FUNCTION "TE-SS" : VOID	// FC 11
AUTHOR : SIMATIC
FAMILY : EA_DIS
NAME : TE_SS
VERSION : 3.0
BEGIN
// (block stored without names or comments; labels and parameter names are numbered)
NETWORK
TITLE =
      L     0;
      L     #PARAM22;
      ==I;
      JC    M001;
      T     MW 214;
      L     MB 214;
      T     LW 10;
      OPN   DB [LW 10];
      L     MB 215;
      SLW   3;
      LAR1;
      L     DBW [AR1,P#0.0];
      T     MB 227;
M001: L     #PARAM20;
      T     MW 214;
      L     MB 214;
      T     LW 10;
      OPN   DB [LW 10];
      L     #PARAM20;
      T     MW 214;
      L     MB 215;
      SLW   3;
      LAR1;
      L     DBW [AR1,P#0.0];
      T     MW 200;
      L     DBW [AR1,P#2.0];
      T     MW 202;
      L     DBW [AR1,P#4.0];
      T     MW 204;
      L     DBW [AR1,P#10.0];
      T     MW 208;
      L     DBW [AR1,P#12.0];
      T     MW 210;
      L     DBW [AR1,P#14.0];
      T     MW 212;
      L     DBW [AR1,P#16.0];
      T     MW 206;
      A     #PARAM1;
      A     M 204.7;
      =     M 203.2;
      A     #PARAM1;
      AN    M 204.7;
      =     M 202.0;
      A     #PARAM2;
      =     M 202.1;
      A     #PARAM3;
      AN    M 203.3;
      =     M 211.5;
      A     #PARAM3;
      =     M 203.3;
      A     #PARAM4;
      AN    M 203.0;
      =     M 211.7;
      A     #PARAM4;
      =     M 203.0;
      A     #PARAM8;
      AN    M 203.1;
      =     M 211.6;
      A     #PARAM8;
      =     M 203.1;
      A     #PARAM9;
      AN    M 203.4;
      =     M 211.4;
      A     #PARAM9;
      =     M 203.4;
      A     #PARAM10;
      =     M 202.2;
      A     #PARAM11;
      =     M 203.5;
      A     #PARAM7;
      =     M 213.0;
      A     #PARAM6;
      =     M 210.1;
      A     #PARAM13;
      =     M 210.7;
      A     #PARAM14;
      =     M 210.6;
      A     #PARAM15;
      =     M 210.5;
      A     #PARAM16;
      =     M 210.4;
      A     #PARAM17;
      =     M 210.3;
      A     #PARAM18;
      =     M 210.2;
      A     #PARAM19;
      =     M 200.4;
      A     #PARAM12;
      =     M 210.0;
      A     #PARAM5;
      =     M 203.6;
NETWORK
TITLE =
      A     M 210.7;
      AN    M 210.6;
      =     M 212.7;
      AN    M 210.7;
      A     M 210.6;
      =     M 212.5;
      A     M 210.5;
      AN    M 210.4;
      =     M 212.6;
      AN    M 210.5;
      A     M 210.4;
      =     M 212.4;
NETWORK
TITLE =
      A     M 227.3;
      AN    M 202.5;
      =     M 211.3;
      A     M 227.3;
      =     M 202.5;
      A     M 227.2;
      AN    M 202.6;
      =     M 211.2;
      A     M 227.2;
      =     M 202.6;
NETWORK
TITLE =
      A     M 203.1;
      A     M 210.1;
      AN    M 203.0;
      AN    M 203.6;
      =     M 218.7;
      A     M 203.0;
      A     M 210.1;
      AN    M 203.6;
      =     M 219.7;
      A     M 227.2;
      A     M 227.1;
      AN    M 227.3;
      AN    M 227.0;
      AN    M 219.7;
      AN    M 203.6;
      =     M 218.5;
      A     M 227.3;
      A     M 227.1;
      AN    M 227.0;
      AN    M 218.7;
      AN    M 203.6;
      =     M 219.5;
      A     M 203.4;
      AN    M 203.3;
      AN    M 219.7;
      AN    M 203.6;
      AN    M 227.0;
      AN    M 219.5;
      =     M 218.3;
      A     M 203.3;
      AN    M 218.7;
      AN    M 218.5;
      AN    M 203.6;
      AN    M 227.0;
      =     M 219.3;
      A     M 218.7;
      O     M 218.5;
      O     M 218.3;
      =     M 212.3;
      A     M 219.7;
      O     M 219.5;
      O     M 219.3;
      =     M 212.1;
      A     M 211.6;
      A     M 218.7;
      O;
      A     M 211.2;
      A     M 218.5;
      O;
      A     M 211.4;
      A     M 218.3;
      =     M 212.2;
      A     M 211.7;
      A     M 219.7;
      O;
      A     M 211.3;
      A     M 219.5;
      O;
      A     M 211.5;
      A     M 219.3;
      =     M 212.0;
NETWORK
TITLE =
      A     M 211.6;
      O     M 211.2;
      =     M 213.4;
      A     M 211.7;
      O     M 211.3;
      =     M 213.5;
      A     M 203.6;
      O     M 227.0;
      =     M 213.7;
NETWORK
TITLE =
      A     M 212.7;
      O     M 213.7;
      O     M 212.3;
      R     M 211.1;
      R     M 211.0;
      A     M 203.2;
      S     M 211.1;
      A     M 202.0;
      S     M 211.0;
      A     M 212.6;
      O     M 213.7;
      O     M 212.1;
      R     M 213.1;
      A     M 203.5;
      S     M 213.1;
NETWORK
TITLE =
      A     M 203.1;
      A     M 210.1;
      O(;
      A     M 227.2;
      A     M 227.1;
      );
      O     M 203.4;
      =     M 213.2;
      A     M 203.0;
      A     M 210.1;
      O(;
      A     M 227.3;
      A     M 227.1;
      );
      O     M 203.3;
      =     M 213.3;
      A     M 213.2;
      O     M 203.5;
      ON    M 202.1;
      A     M 213.3;
      A     M 212.5;
      O(;
      A     M 213.3;
      O     M 203.2;
      O     M 202.0;
      ON    M 202.2;
      A     M 213.2;
      A     M 212.4;
      );
      O(;
      A     M 203.2;
      O     M 202.0;
      A     M 203.5;
      A     M 212.5;
      );
      =     M 201.1;
NETWORK
TITLE =
      L     0;
      L     MW 206;
      >=I;
      JC    M002;
      AN    "M 1.3";
      JC    M002;
      L     MW 206;
      L     1;
      -I;
      T     MW 206;
      L     MB 207;
      T     DBW [AR1,P#16.0];
M002: NOP   0;
NETWORK
TITLE =
      L     MB 205;
      T     MB 209;
      L     0;
      >I;
      JC    M006;
      A     M 212.7;
      A     M 212.4;
      AN    M 204.5;
      O;
      A     M 212.7;
      A     M 212.4;
      A     M 204.5;
      AN    M 210.3;
      L     1;
      JC    M005;
      A     M 212.6;
      A     M 212.5;
      AN    M 204.6;
      O;
      A     M 212.6;
      A     M 212.5;
      A     M 204.6;
      AN    M 210.2;
      L     9;
      JC    M005;
      A     M 212.0;
      A     M 202.1;
      AN    M 213.1;
      O     M 211.1;
      O     M 211.0;
      L     10;
      JC    M003;
      AN    M 212.2;
      ON    M 202.2;
      AN    M 213.1;
      JC    M004;
      L     2;
M003: T     MB 209;
      L     DBW [AR1,P#6.0];
      T     MW 206;
      L     MW 206;
      T     DBW [AR1,P#16.0];
      JU    M006;
M004: L     0;
M005: T     MB 209;
M006: NOP   0;
NETWORK
TITLE =
      L     MB 205;
      L     1;
      <>I;
      JC    M008;
      A     M 212.6;
      O     M 212.5;
      L     14;
      JC    M007;
      A     M 211.0;
      O     M 211.1;
      JC    M008;
      AN    M 212.2;
      ON    M 202.2;
      AN    M 213.1;
      JC    M008;
      L     DBW [AR1,P#6.0];
      T     MW 206;
      L     MW 206;
      T     DBW [AR1,P#16.0];
      L     2;
M007: T     MB 209;
M008: NOP   0;
NETWORK
TITLE =
      L     MB 205;
      L     2;
      <>I;
      JC    M014;
      A     M 212.0;
      A     M 202.1;
      AN    M 213.1;
      O     M 211.0;
      O     M 211.1;
      L     12;
      JC    M009;
      A     M 212.5;
      L     4;
      JC    M012;
      A     M 213.7;
      AN    M 213.1;
      O     M 200.4;
      O;
      AN    M 212.3;
      AN    M 213.0;
      AN    M 213.1;
      L     0;
      JC    M013;
      AN    M 210.2;
      L     6;
      JC    M013;
      L     MW 206;
      L     0;
      <>I;
      JC    M014;
      L     3;
      T     MB 209;
      JU    M014;
M009: T     MB 209;
      L     DBW [AR1,P#6.0];
      JU    M011;
M010: L     DBW [AR1,P#8.0];
M011: T     MW 206;
      T     DBW [AR1,P#16.0];
      JU    M014;
M012: T     MB 209;
      JU    M010;
M013: T     MB 209;
      L     0;
      JU    M011;
M014: NOP   0;
NETWORK
TITLE =
      L     MB 205;
      L     3;
      <>I;
      JC    M017;
      A     M 211.1;
      O     M 200.4;
      O;
      A     M 213.7;
      AN    M 213.1;
      O;
      AN    M 213.0;
      AN    M 212.3;
      AN    M 213.1;
      O;
      A     M 212.0;
      A     M 202.1;
      AN    M 213.1;
      L     0;
      JC    M016;
      A     M 212.7;
      A     M 213.5;
      L     1;
      JC    M016;
      A     M 212.5;
      A     M 213.4;
      L     4;
      JC    M015;
      A     M 210.2;
      L     6;
      JC    M017;
M015: T     MB 209;
      L     DBW [AR1,P#8.0];
      T     MW 206;
      L     MW 206;
      T     DBW [AR1,P#16.0];
      JU    M017;
M016: T     MB 209;
M017: NOP   0;
NETWORK
TITLE =
      L     MB 205;
      L     4;
      <>I;
      JC    M021;
      A     M 212.0;
      A     M 202.1;
      AN    M 213.1;
      O     M 211.0;
      O     M 211.1;
      L     10;
      JC    M018;
      A     M 212.6;
      AN    M 204.6;
      O;
      A     M 212.6;
      A     M 204.6;
      AN    M 210.2;
      L     9;
      JC    M020;
      A     M 213.7;
      AN    M 213.1;
      O     M 200.4;
      O;
      AN    M 212.3;
      AN    M 213.0;
      AN    M 213.1;
      L     0;
      JC    M020;
      AN    M 210.2;
      L     6;
      JC    M020;
      L     MW 206;
      L     0;
      <>I;
      JC    M021;
      L     5;
      T     MB 209;
      JU    M021;
M018: T     MB 209;
      L     DBW [AR1,P#6.0];
M019: T     MW 206;
      L     MW 206;
      T     DBW [AR1,P#16.0];
      JU    M021;
M020: T     MB 209;
      L     0;
      JU    M019;
M021: NOP   0;
NETWORK
TITLE =
      L     MB 205;
      L     5;
      <>I;
      JC    M024;
      A     M 213.7;
      O     M 200.4;
      O;
      AN    M 213.0;
      AN    M 212.3;
      AN    M 213.1;
      L     0;
      JC    M023;
      A     M 212.6;
      AN    M 204.6;
      A     M 213.4;
      O;
      A     M 212.6;
      A     M 204.6;
      AN    M 210.2;
      A     M 213.4;
      L     9;
      JC    M023;
      A     M 211.1;
      O;
      A     M 212.0;
      A     M 202.1;
      AN    M 213.1;
      L     10;
      JC    M022;
      A     M 210.2;
      L     6;
      JC    M024;
M022: T     MB 209;
      L     DBW [AR1,P#6.0];
      T     MW 206;
      L     MW 206;
      T     DBW [AR1,P#16.0];
      JU    M024;
M023: T     MB 209;
M024: NOP   0;
NETWORK
TITLE =
      L     MB 205;
      L     6;
      <>I;
      JC    M025;
      AN    M 213.5;
      AN    M 213.4;
      L     0;
      JC    M025;
      T     MB 209;
M025: NOP   0;
NETWORK
TITLE =
      L     MB 205;
      L     9;
      <>I;
      JC    M027;
      A     M 212.7;
      O     M 212.4;
      O     M 200.4;
      L     6;
      JC    M026;
      AN    M 211.0;
      AN    M 211.1;
      A(;
      AN    M 212.0;
      ON    M 202.1;
      O     M 213.1;
      );
      JC    M027;
      L     DBW [AR1,P#6.0];
      T     MW 206;
      L     MW 206;
      T     DBW [AR1,P#0.0];
      L     10;
M026: T     MB 209;
M027: NOP   0;
NETWORK
TITLE =
      L     MB 205;
      L     10;
      <>I;
      JC    M033;
      A     M 212.2;
      A     M 202.2;
      O     M 213.1;
      AN    M 211.0;
      AN    M 211.1;
      L     4;
      JC    M028;
      A     M 212.4;
      L     12;
      JC    M031;
      A     M 213.7;
      AN    M 211.1;
      AN    M 211.0;
      O     M 200.4;
      O;
      AN    M 212.1;
      AN    M 213.0;
      AN    M 211.1;
      AN    M 211.0;
      L     0;
      JC    M032;
      AN    M 210.3;
      L     14;
      JC    M032;
      L     MW 206;
      L     0;
      <>I;
      JC    M033;
      L     11;
      T     MB 209;
      JU    M033;
M028: T     MB 209;
      L     DBW [AR1,P#6.0];
      JU    M030;
M029: L     DBW [AR1,P#8.0];
M030: T     MW 206;
      L     MW 206;
      T     DBW [AR1,P#16.0];
      JU    M033;
M031: T     MB 209;
      JU    M029;
M032: T     MB 209;
      L     0;
      JU    M030;
M033: NOP   0;
NETWORK
TITLE =
      L     MB 205;
      L     11;
      <>I;
      JC    M036;
      A     M 200.4;
      O;
      A     M 213.7;
      AN    M 211.1;
      AN    M 211.0;
      O;
      AN    M 213.0;
      AN    M 212.1;
      AN    M 211.1;
      AN    M 211.0;
      O;
      A     M 212.2;
      A     M 202.2;
      AN    M 211.1;
      AN    M 211.0;
      L     0;
      JC    M035;
      A     M 212.6;
      A     M 213.4;
      L     9;
      JC    M035;
      A     M 212.4;
      A     M 213.5;
      L     12;
      JC    M034;
      A     M 210.3;
      L     14;
      JC    M036;
M034: T     MB 209;
      L     DBW [AR1,P#8.0];
      T     MW 206;
      L     MW 206;
      T     DBW [AR1,P#16.0];
      JU    M036;
M035: T     MB 209;
M036: NOP   0;
NETWORK
TITLE =
      L     MB 205;
      L     12;
      <>I;
      JC    M040;
      A     M 212.2;
      A     M 202.2;
      O     M 213.1;
      AN    M 211.0;
      AN    M 211.1;
      L     2;
      JC    M037;
      A     M 212.7;
      AN    M 204.5;
      O;
      A     M 212.7;
      A     M 204.5;
      AN    M 210.3;
      =     M 228.0;
      A     M 228.0;
      A     M 211.1;
      L     6;
      JC    M039;
      A     M 228.0;
      L     1;
      JC    M039;
      A     M 213.7;
      AN    M 211.1;
      AN    M 211.0;
      O     M 200.4;
      O;
      AN    M 212.1;
      AN    M 213.0;
      AN    M 211.1;
      AN    M 211.0;
      L     0;
      JC    M039;
      AN    M 210.3;
      L     14;
      JC    M039;
      L     MW 206;
      L     0;
      <>I;
      JC    M040;
      L     13;
      T     MB 209;
      JU    M040;
M037: T     MB 209;
      L     DBW [AR1,P#6.0];
M038: T     MW 206;
      L     MW 206;
      T     DBW [AR1,P#16.0];
      JU    M040;
M039: T     MB 209;
      L     0;
      JU    M038;
M040: NOP   0;
NETWORK
TITLE =
      L     MB 205;
      L     13;
      <>I;
      JC    M043;
      A     M 213.7;
      O     M 200.4;
      O;
      AN    M 213.0;
      AN    M 212.1;
      AN    M 211.1;
      AN    M 211.0;
      L     0;
      JC    M042;
      A     M 212.7;
      AN    M 204.5;
      A     M 213.5;
      O;
      A     M 212.7;
      A     M 204.5;
      AN    M 210.3;
      A     M 213.5;
      L     1;
      JC    M042;
      A     M 212.2;
      A     M 202.2;
      AN    M 211.1;
      AN    M 211.0;
      L     2;
      JC    M041;
      A     M 210.3;
      L     14;
      JC    M043;
M041: T     MB 209;
      L     DBW [AR1,P#6.0];
      T     MW 206;
      L     MW 206;
      T     DBW [AR1,P#16.0];
      JU    M043;
M042: T     MB 209;
M043: NOP   0;
NETWORK
TITLE =
      L     MB 205;
      L     14;
      <>I;
      JC    M044;
      AN    M 213.5;
      AN    M 213.4;
      L     0;
      JC    M044;
      T     MB 209;
M044: NOP   0;
NETWORK
TITLE =
      L     MB 209;
      T     MB 205;
      L     15;
      <I;
      A(;
      +     -7;
      <>I;
      );
      A(;
      +     -1;
      <>I;
      );
      AN    "M 0.7";
      JC    M045;
      L     0;
      T     MB 205;
M045: NOP   0;
NETWORK
TITLE =
      A     M 212.6;
      A     M 212.7;
      O;
      AN    M 212.6;
      AN    M 212.4;
      O;
      AN    M 212.7;
      AN    M 212.5;
      =     M 200.7;
      AN    M 210.2;
      AN    M 210.3;
      =     M 202.7;
      A     M 212.6;
      AN    M 210.2;
      =     M 200.5;
      A     M 212.7;
      AN    M 210.3;
      =     M 200.6;
      AN    M 209.0;
      A     M 209.1;
      A     M 209.2;
      AN    M 200.7;
      =     M 228.0;
      AN    M 209.3;
      A     M 228.0;
      =     M 200.2;
      A     M 209.3;
      A     M 228.0;
      =     M 200.3;
      A     M 209.0;
      A(;
      A     M 209.1;
      AN    M 209.2;
      O;
      AN    M 209.1;
      A     M 209.2;
      );
      AN    M 200.7;
      AN    M 202.7;
      =     M 228.0;
      A     M 228.0;
      AN    M 209.3;
      =     M 200.1;
      A     M 228.0;
      A     M 209.3;
      =     M 200.0;
NETWORK
TITLE =
      A     M 201.1;
      =     M 203.7;
      A     M 209.0;
      A     M 209.1;
      A     M 209.2;
      O     M 200.4;
      O     M 200.3;
      O     M 200.2;
      O     M 200.1;
      O     M 200.0;
      O     M 200.7;
      O     M 202.7;
      =     M 201.0;
      A(;
      A     M 209.1;
      AN    M 209.2;
      O;
      AN    M 209.1;
      A     M 209.2;
      );
      AN    M 209.0;
      =     M 228.0;
      A     M 228.0;
      A     M 209.3;
      =     M 201.4;
      A     M 200.0;
      O     M 200.3;
      AN    M 200.7;
      AN    M 202.7;
      =     M 201.2;
      A     M 212.7;
      AN    M 204.5;
      O;
      A     M 212.7;
      A     M 204.5;
      AN    M 210.3;
      =     M 201.3;
      =     M 202.4;
      =     #PARAM24;
      A     M 228.0;
      AN    M 209.3;
      =     M 201.7;
      A     M 200.1;
      O     M 200.2;
      AN    M 200.7;
      AN    M 202.7;
      =     M 201.5;
      A     M 212.6;
      AN    M 204.6;
      O;
      A     M 212.6;
      AN    M 210.2;
      A     M 204.6;
      =     M 201.6;
      =     M 202.3;
      =     #PARAM25;
NETWORK
TITLE =
      A     M 201.0;
      O     M 203.7;
      AN    M 201.1;
      =     #PARAM26;
      A     M 201.0;
      A     "M 1.6";
      O     M 203.7;
      O     #PARAM12;
      =     #PARAM29;
      A     M 201.7;
      A     "M 1.5";
      O;
      A     M 201.5;
      A     "M 1.6";
      O     M 201.6;
      O     #PARAM12;
      =     #PARAM28;
      A     M 201.4;
      A     "M 1.5";
      O;
      A     M 201.2;
      A     "M 1.6";
      O     M 201.3;
      O     #PARAM12;
      =     #PARAM27;
NETWORK
TITLE =
      A(;
      A     M 209.1;
      AN    M 209.2;
      O;
      AN    M 209.1;
      A     M 209.2;
      );
      AN    M 209.3;
      =     #PARAM31;
      A(;
      A     M 209.1;
      AN    M 209.2;
      O;
      AN    M 209.1;
      A     M 209.2;
      );
      A     M 209.3;
      =     #PARAM30;
      L     MW 200;
      T     DBW [AR1,P#0.0];
      L     MW 202;
      T     DBW [AR1,P#2.0];
      L     MW 204;
      T     DBW [AR1,P#4.0];
      L     MW 208;
      T     DBW [AR1,P#10.0];
      L     MW 210;
      T     DBW [AR1,P#12.0];
      L     MW 212;
      T     DBW [AR1,P#14.0];
      L     MW 206;
      T     DBW [AR1,P#16.0];
      L     0;
      L     #PARAM23;
      ==I;
      JC    M048;
      T     MW 216;
      T     MW 240;
      L     MB 216;
      SLW   3;
      LAR1;
      L     DBW [AR1,P#0.0];
      T     MW 242;
      L     MW 240;
      SLW   12;
      SRW   12;
      T     MW 240;
      L     8;
      L     MB 241;
      >I;
      JC    M046;
      +     -8;
      SLW   8;
      INC   242;
      JU    M047;
M046: SLW   8;
      INC   243;
M047: T     MW 244;
      L     MB 244;
      L     MB 245;
      SLW   3;
      OW;
      LAR2;
      A     M 201.0;
      O     M 203.3;
      =     M [AR2,P#0.0];
      L     MB 217;
      SLW   3;
      LAR1;
      L     MW 242;
      T     DBW [AR1,P#0.0];
M048: L     0;
      L     #PARAM21;
      ==I;
      BEC;
      T     MW 216;
      L     MB 216;
      T     LW 10;
      OPN   DB [LW 10];
      L     MB 217;
      SLW   3;
      LAR1;
      L     MW 200;
      T     DBW [AR1,P#0.0];
      L     MW 202;
      T     DBW [AR1,P#2.0];
END_FUNCTION

FUNCTION "TE-REK" : VOID	// FC 12
AUTHOR : SIMATIC
FAMILY : SIMATIC
NAME : TE_REK
VERSION : 3.0
BEGIN
// (block stored without names or comments; labels and parameter names are numbered)
NETWORK
TITLE =
      L     0;
      L     #PARAM20;
      ==I;
      JC    M001;
      T     MW 212;
      L     MB 212;
      T     LW 10;
      OPN   DB [LW 10];
      L     MB 213;
      SLW   3;
      LAR1;
      L     DBW [AR1,P#2.0];
M001: T     MW 210;
      L     #PARAM18;
      T     MW 214;
      L     MB 214;
      T     LW 10;
      OPN   DB [LW 10];
      L     MB 215;
      SLW   3;
      LAR1;
      L     DBW [AR1,P#0.0];
      T     MW 200;
      L     DBW [AR1,P#2.0];
      T     MW 202;
      A     #PARAM1;
      =     M 203.1;
      A     #PARAM2;
      =     M 200.4;
      A     #PARAM3;
      AN    M 202.7;
      =     M 210.0;
      A     #PARAM3;
      =     M 202.7;
      A     #PARAM4;
      AN    M 200.2;
      =     M 210.1;
      A     #PARAM4;
      =     M 200.2;
      A     #PARAM6;
      AN    M 200.3;
      =     M 210.3;
      A     #PARAM6;
      =     M 200.3;
      A     #PARAM7;
      AN    M 202.6;
      =     M 210.2;
      A     #PARAM7;
      =     M 202.6;
      A     #PARAM8;
      =     M 200.5;
      A     #PARAM9;
      =     M 203.0;
      A     #PARAM10;
      =     M 210.7;
      A     #PARAM5;
      =     M 202.5;
      A     #PARAM11;
      AN    M 200.0;
      =     M 210.4;
      A     #PARAM11;
      =     M 200.0;
      A     #PARAM12;
      AN    M 200.1;
      =     M 210.5;
      A     #PARAM12;
      =     M 200.1;
      A     #PARAM13;
      AN    M 202.4;
      =     M 210.6;
      A     #PARAM13;
      =     M 202.4;
      AN    #PARAM14;
      =     M 200.6;
      A     #PARAM15;
      =     M 203.3;
NETWORK
TITLE =
      A     M 211.0;
      AN    M 202.3;
      =     M 211.5;
      A     M 211.0;
      =     M 202.3;
      A     M 211.2;
      AN    M 202.1;
      =     M 211.6;
      A     M 211.2;
      =     M 202.1;
      A     M 211.3;
      AN    M 202.2;
      =     M 211.7;
      A     M 211.3;
      =     M 202.2;
NETWORK
TITLE =
      AN    M 200.7;
      AN    M 201.5;
      S     M 200.7;
      A     "´1´";
      R     M 201.7;
      R     M 201.6;
NETWORK
TITLE =
      A     M 202.7;
      A     M 202.5;
      O;
      A     M 202.1;
      A     M 211.1;
      O;
      A     M 200.2;
      =     M 202.0;
      A     M 202.6;
      A     M 202.5;
      O;
      A     M 202.2;
      A     M 211.1;
      O;
      A     M 200.3;
      =     M 203.6;
NETWORK
TITLE =
      AN    M 200.7;
      JC    M005;
      AN    M 203.1;
      JC    M002;
      L     MW 214;
      +     5;
      T     MW 216;
      +     -2;
      T     MW 218;
      L     DBW [AR1,P#10.0];
      T     DBW [AR1,P#6.0];
      JU    M005;
M002: AN    M 203.0;
      JC    M003;
      L     MW 214;
      +     6;
      T     MW 216;
      +     -3;
      T     MW 218;
      L     DBW [AR1,P#12.0];
      T     DBW [AR1,P#6.0];
      JU    M008;
M003: A     M 211.5;
      A     M 211.1;
      AN    M 202.4;
      O;
      A     M 210.6;
      A     M 202.5;
      AN    M 211.0;
      S     M 201.7;
      A     M 210.5;
      AN    M 200.0;
      O     M 201.7;
      O     M 211.5;
      R     M 200.7;
      S     M 201.5;
      R     M 210.5;
      R     M 211.5;
      R     M 210.6;
      A     M 202.0;
      AN    M 203.6;
      A     M 200.4;
      S     M 203.5;
      AN    M 202.0;
      R     M 203.5;
      A     M 203.6;
      AN    M 202.0;
      A     M 200.5;
      S     M 203.4;
      AN    M 203.6;
      R     M 203.4;
      AN    M 203.5;
      JC    M006;
      L     MW 214;
      +     2;
      T     MW 216;
      L     DBW [AR1,P#4.0];
      T     MW 206;
      SLW   6;
      SRW   6;
      L     DBB [AR1,P#4.0];
      SRW   2;
      +I;
      L     1000;
      TAK;
      >I;
      JC    M004;
      TAK;
M004: T     MW 204;
      L     MB 206;
      SRW   2;
      SLW   10;
      OW;
      T     DBW [AR1,P#4.0];
      L     MW 214;
      +     3;
      T     MW 216;
      L     DBW [AR1,P#6.0];
      L     MW 204;
      -I;
      T     DBW [AR1,P#6.0];
M005: JU    M008;
M006: AN    M 203.4;
      JC    M009;
      L     MW 214;
      +     2;
      T     MW 216;
      L     DBW [AR1,P#4.0];
      T     MW 206;
      SLW   6;
      SRW   6;
      L     DBB [AR1,P#4.0];
      SRW   2;
      +I;
      L     1000;
      TAK;
      >I;
      JC    M007;
      TAK;
M007: T     MW 204;
      L     MB 206;
      SRW   2;
      SLW   10;
      OW;
      T     DBW [AR1,P#4.0];
      L     MW 214;
      +     3;
      T     MW 216;
      L     DBW [AR1,P#6.0];
      L     MW 204;
      +I;
      T     DBW [AR1,P#6.0];
M008: JU    M010;
M009: L     MW 214;
      +     2;
      T     MW 216;
      L     DBB [AR1,P#4.0];
      SRW   2;
      SLW   10;
      T     DBW [AR1,P#4.0];
      L     0;
      L     #PARAM20;
      ==I;
      JC    M010;
      T     MW 212;
      L     MW 214;
      +     8;
      T     MW 216;
      L     DBW [AR1,P#16.0];
      T     LD 0;
      L     MB 212;
      T     LW 10;
      OPN   DB [LW 10];
      L     MB 213;
      SLW   3;
      LAR1;
      L     LD 0;
      L     DBW [AR1,P#0.0];
      ==I;
      T     LD 0;
      L     MB 214;
      T     LW 10;
      OPN   DB [LW 10];
      JC    M010;
      L     MB 215;
      SLW   3;
      LAR1;
      L     LD 0;
      T     DBW [AR1,P#16.0];
      L     MW 214;
      +     3;
      T     MW 216;
      L     LD 0;
      T     DBW [AR1,P#6.0];
M010: NOP   0;
NETWORK
TITLE =
      AN    M 201.5;
      JC    M013;
      AN    M 203.1;
      JC    M011;
      L     MW 214;
      +     5;
      T     MW 216;
      +     -2;
      T     MW 218;
      L     MB 215;
      SLW   3;
      LAR1;
      L     DBW [AR1,P#10.0];
      T     DBW [AR1,P#6.0];
      JU    M012;
M011: AN    M 203.0;
      JC    M012;
      L     MW 214;
      +     6;
      T     MW 216;
      +     -3;
      T     MW 218;
      L     MB 215;
      SLW   3;
      LAR1;
      L     DBW [AR1,P#12.0];
      T     DBW [AR1,P#6.0];
M012: A     M 211.5;
      A     M 211.1;
      AN    M 202.4;
      O;
      A     M 210.6;
      A     M 202.5;
      AN    M 211.0;
      S     M 201.6;
      A     M 210.4;
      AN    M 200.1;
      AN    M 202.4;
      AN    M 202.3;
      O     M 211.5;
      O     M 201.6;
      O     M 200.6;
      O     "M 0.6";
      O     M 203.3;
      S     M 200.7;
      R     M 201.5;
      A     M 200.7;
      O     M 203.0;
      O     M 203.1;
      JC    M013;
      L     #PARAM16;
      T     MW 216;
      L     MB 216;
      T     LW 10;
      OPN   DB [LW 10];
      L     MB 217;
      SLW   3;
      LAR1;
      L     DBD [AR1,P#0.0];
      T     LD 0;
      L     MB 214;
      T     LW 10;
      OPN   DB [LW 10];
      L     MW 214;
      +     3;
      T     MW 216;
      L     MB 215;
      SLW   3;
      LAR1;
      L     LW 8;
      L     LD 0;
      T     DBD [AR1,P#18.0];
M013: NOP   0;
NETWORK
TITLE =
      L     MW 214;
      +     3;
      T     MW 216;
      +     4;
      T     MW 218;
      L     MB 215;
      SLW   3;
      LAR1;
      L     DBW [AR1,P#6.0];
      L     DBW [AR1,P#14.0];
      ==I;
      T     MW 222;
      JC    M019;
      <=I;
      JC    M016;
      AN    M 200.5;
      AN    M 203.0;
      JC    M019;
      TAK;
      T     MW 224;
      L     MW 214;
      +     6;
      T     MW 216;
      L     DBW [AR1,P#12.0];
      L     DBW [AR1,P#10.0];
      -I;
      SRW   3;
      L     MW 222;
      +I;
      L     MW 224;
      <=I;
      TAK;
      JC    M014;
      TAK;
M014: T     MW 222;
      L     MW 214;
      +     6;
      T     MW 216;
      L     DBW [AR1,P#12.0];
      L     MW 222;
      >I;
      JC    M015;
      L     MW 214;
      +     3;
      T     MW 216;
      L     DBW [AR1,P#12.0];
      T     DBW [AR1,P#6.0];
M015: NOP   0;
      T     DBW [AR1,P#14.0];
      T     MW 222;
      L     MW 218;
      +     2;
      T     MW 218;
      TAK;
      L     MW 222;
      L     1;
      *I;
      DTR;
      T     DBD [AR1,P#18.0];
      JU    M019;
M016: ==I;
      JC    M019;
      AN    M 200.4;
      AN    M 203.1;
      JC    M019;
      TAK;
      T     MW 224;
      L     MW 214;
      +     6;
      T     MW 216;
      L     DBW [AR1,P#12.0];
      L     DBW [AR1,P#10.0];
      -I;
      SRW   3;
      L     MW 222;
      TAK;
      -I;
      L     MW 224;
      >=I;
      TAK;
      JC    M017;
      TAK;
M017: T     MW 222;
      L     MW 214;
      +     5;
      T     MW 216;
      L     DBW [AR1,P#10.0];
      L     MW 222;
      <I;
      JC    M018;
      L     MW 214;
      +     3;
      T     MW 216;
      L     DBW [AR1,P#10.0];
      T     DBW [AR1,P#6.0];
M018: NOP   0;
      T     DBW [AR1,P#14.0];
      T     MW 222;
      L     1;
      *I;
      DTR;
      T     DBD [AR1,P#18.0];
M019: NOP   0;
NETWORK
TITLE =
      A(;
      A     M 203.0;
      O     M 203.1;
      ON    M 200.5;
      ON    M 200.4;
      A     M 201.5;
      );
      O(;
      A(;
      O     M 202.4;
      O     M 202.3;
      );
      A(;
      O     M 200.6;
      O     M 203.3;
      );
      );
      O(;
      A     M 203.0;
      ON    M 200.4;
      A     M 202.0;
      A     M 200.7;
      );
      O(;
      A     M 203.1;
      ON    M 200.5;
      A     M 203.6;
      A     M 200.7;
      );
      =     M 201.3;
      A     M 203.5;
      O     M 203.4;
      O     M 203.0;
      O     M 203.1;
      =     M 203.7;
      =     M 203.2;
NETWORK
TITLE =
// (network holds code this reader does not know; not shown)
END_FUNCTION

FUNCTION "TE-TS" : VOID	// FC 13
AUTHOR : SIMATIC
FAMILY : EA_DIS
NAME : TE_TS
VERSION : 3.0
BEGIN
// (block stored without names or comments; labels and parameter names are numbered)
NETWORK
TITLE =
      L     0;
      L     #PARAM9;
      ==I;
      JC    M001;
      T     MW 212;
      L     MB 212;
      T     LW 10;
      OPN   DB [LW 10];
      L     MB 213;
      SLW   3;
      LAR1;
      L     DBW [AR1,P#0.0];
      T     MB 207;
M001: OPN   #PARAM6;
      L     #PARAM7;
      T     MW 212;
      L     MB 213;
      SLW   3;
      LAR1;
      L     DBW [AR1,P#0.0];
      T     MW 200;
      A     #PARAM1;
      AN    M 201.5;
      =     M 203.5;
      A     #PARAM1;
      =     M 201.5;
      A     #PARAM2;
      AN    M 201.6;
      =     M 203.6;
      A     #PARAM2;
      =     M 201.6;
      A     #PARAM3;
      AN    M 201.4;
      =     M 203.4;
      A     #PARAM3;
      =     M 201.4;
      A     #PARAM4;
      =     M 201.3;
      A     #PARAM5;
      =     M 200.7;
NETWORK
TITLE =
      A     M 207.0;
      A     M 207.1;
      AN    M 200.0;
      =     M 203.0;
      A     M 207.0;
      =     M 200.0;
NETWORK
TITLE =
      A     M 207.3;
      AN    M 200.3;
      =     M 203.3;
      A     M 207.3;
      =     M 200.3;
NETWORK
TITLE =
      A     M 207.2;
      AN    M 200.2;
      =     M 203.2;
      A     M 207.2;
      =     M 200.2;
NETWORK
TITLE =
      A     M 203.0;
      A     M 207.1;
      A     M 201.7;
      =     M 203.1;
      A     M 203.0;
      A     M 207.1;
      AN    M 201.7;
      =     M 203.7;
      A     M 203.6;
      A     M 201.3;
      A     M 201.7;
      =     M 202.0;
      A     M 203.6;
      A     M 201.3;
      AN    M 201.7;
      =     M 202.1;
NETWORK
TITLE =
      A     M 200.2;
      A     M 207.1;
      O;
      A     M 201.7;
      A     M 200.0;
      A     M 207.1;
      O;
      A     M 201.7;
      A     M 201.6;
      A     M 201.3;
      O     M 201.5;
      =     M 200.5;
      A     M 200.3;
      A     M 207.1;
      O;
      AN    M 201.7;
      A     M 200.0;
      A     M 207.1;
      O;
      AN    M 201.7;
      A     M 201.6;
      A     M 201.3;
      O     M 201.4;
      =     M 200.6;
NETWORK
TITLE =
      A(;
      A     M 203.3;
      AN    M 200.2;
      O     M 203.7;
      O     M 202.1;
      O     M 201.4;
      );
      S     M 201.7;
      A(;
      A     M 203.2;
      AN    M 200.3;
      O     M 203.1;
      O     M 202.0;
      );
      AN    M 201.4;
      O     M 201.5;
      R     M 201.7;
NETWORK
TITLE =
      A     M 201.7;
      =     M 201.2;
      =     #PARAM11;
      AN    M 201.7;
      =     M 201.1;
      =     #PARAM12;
      A     M 200.6;
      A     M 200.5;
      =     M 201.0;
NETWORK
TITLE =
      A     M 201.0;
      O     M 200.7;
      =     #PARAM14;
      A     M 201.1;
      O     M 200.7;
      =     #PARAM13;
      A     M 201.2;
      O     M 200.7;
      =     #PARAM15;
NETWORK
TITLE =
      L     MW 200;
      T     DBW [AR1,P#0.0];
      L     0;
      L     #PARAM10;
      ==I;
      JC    M004;
      T     MW 212;
      T     MW 220;
      L     MB 212;
      SLW   3;
      LAR1;
      L     DBW [AR1,P#2.0];
      T     MW 208;
      L     MW 220;
      SLW   12;
      SRW   12;
      T     MW 220;
      L     8;
      L     MB 221;
      >I;
      JC    M002;
      +     -8;
      SLW   8;
      INC   208;
      JU    M003;
M002: SLW   8;
      INC   209;
M003: T     MW 210;
      L     MB 210;
      L     MB 211;
      SLW   3;
      OW;
      LAR2;
      A     M 201.0;
      =     M [AR2,P#0.0];
      L     MB 212;
      SLW   3;
      LAR1;
      L     MW 208;
      T     DBW [AR1,P#2.0];
M004: L     0;
      L     #PARAM8;
      ==I;
      JC    M005;
      T     MW 214;
      L     MB 214;
      T     LW 10;
      OPN   DB [LW 10];
      L     MB 215;
      SLW   3;
      LAR1;
      L     MW 200;
      T     DBW [AR1,P#0.0];
M005: NOP   0;
END_FUNCTION

FUNCTION "TE-VW3/3" : VOID	// FC 14
AUTHOR : SIMATIC
FAMILY : EA_DIS
NAME : TE_VW3_3
VERSION : 3.0
BEGIN
// (block stored without names or comments; labels and parameter names are numbered)
NETWORK
TITLE =
      L     0;
      L     #PARAM14;
      ==I;
      JC    M001;
      T     MW 212;
      L     MB 212;
      T     LW 10;
      OPN   DB [LW 10];
      L     MB 213;
      SLW   3;
      LAR1;
      L     DBW [AR1,P#0.0];
      T     MB 203;
M001: L     #PARAM12;
      T     MW 214;
      L     MB 214;
      T     LW 10;
      OPN   DB [LW 10];
      L     MB 215;
      SLW   3;
      LAR1;
      L     DBW [AR1,P#0.0];
      T     MW 200;
      L     DBW [AR1,P#2.0];
      T     MB 202;
      A     #PARAM1;
      =     M 200.0;
      A     #PARAM2;
      AN    M 201.7;
      =     M 204.5;
      A     #PARAM2;
      =     M 201.7;
      A     #PARAM3;
      AN    M 200.1;
      =     M 205.4;
      A     #PARAM3;
      =     M 200.1;
      A     #PARAM4;
      =     M 200.3;
      A     #PARAM5;
      AN    M 200.2;
      =     M 204.6;
      A     #PARAM5;
      =     M 200.2;
      A     #PARAM6;
      AN    M 200.4;
      =     M 205.5;
      A     #PARAM6;
      =     M 200.4;
      A     #PARAM7;
      =     M 200.6;
      A     #PARAM8;
      AN    M 200.5;
      =     M 204.7;
      A     #PARAM8;
      =     M 200.5;
      A     #PARAM9;
      AN    M 200.7;
      =     M 205.6;
      A     #PARAM9;
      =     M 200.7;
      A     #PARAM10;
      =     M 201.6;
      A     #PARAM11;
      =     M 201.5;
NETWORK
TITLE =
      A     M 203.0;
      AN    M 202.0;
      =     M 204.0;
      A     M 203.0;
      =     M 202.0;
      A     M 203.1;
      AN    M 202.1;
      =     M 204.1;
      A     M 203.1;
      =     M 202.1;
      A     M 203.2;
      AN    M 202.2;
      =     M 204.2;
      A     M 203.2;
      =     M 202.2;
NETWORK
TITLE =
      A(;
      A     M 205.4;
      A     M 201.6;
      O;
      A     M 204.0;
      AN    M 200.4;
      AN    M 200.7;
      O;
      A     M 204.5;
      AN    M 200.4;
      AN    M 200.7;
      AN    M 203.1;
      AN    M 203.2;
      );
      A     M 200.0;
      =     M 202.5;
      A(;
      A     M 205.5;
      A     M 201.6;
      O;
      A     M 204.1;
      AN    M 200.1;
      AN    M 200.7;
      O;
      A     M 204.6;
      AN    M 200.1;
      AN    M 200.7;
      AN    M 203.0;
      AN    M 203.2;
      );
      A     M 200.3;
      =     M 202.6;
      A(;
      A     M 205.6;
      A     M 201.6;
      O;
      A     M 204.2;
      AN    M 200.4;
      AN    M 200.1;
      O;
      A     M 204.7;
      AN    M 200.4;
      AN    M 200.1;
      AN    M 203.1;
      AN    M 203.0;
      );
      A     M 200.6;
      =     M 202.7;
NETWORK
TITLE =
      AN    M 201.1;
      AN    M 201.2;
      S     M 201.0;
      A     "´1´";
      S     M 201.3;
      R     M 201.4;
NETWORK
TITLE =
      AN    M 201.0;
      JC    M002;
      A     M 202.6;
      S     M 201.1;
      R     M 201.0;
      A     M 202.7;
      S     M 201.2;
      R     M 201.0;
M002: NOP   0;
NETWORK
TITLE =
      AN    M 201.1;
      JC    M003;
      A     M 202.5;
      S     M 201.0;
      R     M 201.1;
      A     M 202.7;
      S     M 201.2;
      R     M 201.1;
M003: NOP   0;
NETWORK
TITLE =
      AN    M 201.2;
      JC    M004;
      A     M 202.6;
      S     M 201.1;
      R     M 201.2;
      A     M 202.5;
      S     M 201.0;
      R     M 201.2;
M004: NOP   0;
NETWORK
TITLE =
      A     M 201.0;
      =     #PARAM15;
      A     M 201.1;
      =     #PARAM16;
      A     M 201.2;
      =     #PARAM17;
      A     M 201.0;
      O     M 201.5;
      =     #PARAM18;
      A     M 201.1;
      O     M 201.5;
      =     #PARAM19;
      A     M 201.2;
      O     M 201.5;
      =     #PARAM20;
      L     MW 200;
      T     DBW [AR1,P#0.0];
      L     MW 202;
      T     DBW [AR1,P#2.0];
      L     0;
      L     #PARAM13;
      ==I;
      BEC;
      T     MW 216;
      L     MB 216;
      T     LW 10;
      OPN   DB [LW 10];
      L     MB 217;
      SLW   3;
      LAR1;
      L     MB 201;
      T     DBW [AR1,P#0.0];
END_FUNCTION

FUNCTION "TE-KO" : VOID	// FC 15
AUTHOR : SIMATIC
FAMILY : EA_DIS
NAME : TE_KO
VERSION : 0.0
BEGIN
// (block stored without names or comments; labels and parameter names are numbered)
NETWORK
TITLE =
      L     0;
      L     #PARAM18;
      ==I;
      JC    M001;
      T     MW 214;
      L     MB 214;
      T     LW 10;
      OPN   DB [LW 10];
      L     MB 215;
      SLW   3;
      LAR1;
      L     DBW [AR1,P#0.0];
      T     MB 230;
M001: L     #PARAM16;
      T     MW 214;
      L     MB 214;
      T     LW 10;
      OPN   DB [LW 10];
      L     #PARAM16;
      T     MW 214;
      L     MB 215;
      SLW   3;
      LAR1;
      L     DBW [AR1,P#8.0];
      T     MB 203;
      L     DBW [AR1,P#12.0];
      T     MB 209;
      L     DBW [AR1,P#16.0];
      T     MB 212;
      A     #PARAM1;
      =     M 202.0;
      =     #PARAM22;
      A     #PARAM2;
      =     M 203.4;
      A     #PARAM3;
      AN    M 212.2;
      =     M 220.3;
      A     #PARAM3;
      =     M 212.2;
      A     #PARAM4;
      AN    M 203.2;
      =     M 220.1;
      A     #PARAM4;
      =     M 203.2;
      A     #PARAM5;
      =     M 202.2;
      =     #PARAM23;
      A     #PARAM6;
      AN    M 203.0;
      =     M 221.6;
      A     #PARAM6;
      =     M 203.0;
      A     #PARAM7;
      AN    M 212.0;
      =     M 220.2;
      A     #PARAM7;
      =     M 212.0;
      A     #PARAM9;
      AN    M 203.1;
      =     M 221.7;
      A     #PARAM9;
      =     M 203.1;
      A     #PARAM10;
      =     M 202.3;
      =     #PARAM28;
      A     #PARAM11;
      AN    M 203.3;
      =     M 220.0;
      A     #PARAM11;
      =     M 203.3;
      A     #PARAM12;
      AN    M 212.3;
      =     M 220.4;
      A     #PARAM12;
      =     M 212.3;
      A     #PARAM13;
      =     M 203.5;
      A     #PARAM14;
      =     M 202.1;
      =     #PARAM29;
      A     #PARAM8;
      =     M 221.5;
      A     #PARAM15;
      =     M 221.4;
NETWORK
TITLE =
      A     M 230.0;
      AN    M 212.4;
      =     M 220.5;
      A     M 230.0;
      =     M 212.4;
      A     M 230.4;
      AN    M 212.6;
      =     M 220.6;
      A     M 230.4;
      =     M 212.6;
      A     M 230.5;
      AN    M 212.7;
      =     M 220.7;
      A     M 230.5;
      =     M 212.7;
NETWORK
TITLE =
      A(;
      A     M 220.2;
      A     M 221.5;
      O;
      A     M 220.5;
      A     M 230.1;
      );
      =     M 232.1;
      AN    M 232.1;
      AN    M 221.7;
      AN    M 221.6;
      JC    M002;
      A     M 221.7;
      AN    M 203.0;
      O     M 232.1;
      AN    M 209.0;
      S     M 209.0;
      R     M 232.1;
      A     M 221.6;
      O     M 232.1;
      A     M 209.0;
      R     M 209.0;
M002: NOP   0;
NETWORK
TITLE =
      A(;
      A     M 220.4;
      A     M 221.5;
      O;
      A     M 220.7;
      A     M 230.1;
      AN    M 230.4;
      O;
      A     M 220.0;
      AN    M 203.2;
      AN    M 230.4;
      );
      AN    M 212.2;
      =     M 221.3;
NETWORK
TITLE =
      A(;
      A     M 220.3;
      A     M 221.5;
      O;
      A     M 220.6;
      A     M 230.1;
      AN    M 212.3;
      O;
      A     M 220.1;
      AN    M 212.3;
      AN    M 230.5;
      );
      =     M 221.2;
NETWORK
TITLE =
      A     M 212.3;
      A     M 221.5;
      O;
      A     M 230.5;
      A     M 230.1;
      O;
      A     M 203.3;
      =     M 221.1;
      A     M 212.2;
      A     M 221.5;
      O;
      A     M 230.4;
      A     M 230.1;
      O;
      A     M 203.2;
      =     M 221.0;
      A(;
      A(;
      AN    M 203.5;
      O     M 202.0;
      A     M 221.0;
      A     M 203.4;
      );
      A     M 221.1;
      );
      O(;
      A(;
      AN    M 203.4;
      O     M 202.1;
      A     M 221.1;
      A     M 203.5;
      );
      A     M 221.0;
      );
      O(;
      A     M 203.0;
      A     M 203.1;
      );
      =     M 200.1;
NETWORK
TITLE =
      A     M 209.0;
      =     #PARAM26;
      JC    M003;
      R     M 212.1;
      R     M 212.5;
      R     M 209.3;
      R     M 209.4;
M003: NOP   0;
NETWORK
TITLE =
      AN    M 209.0;
      =     #PARAM25;
      JC    M004;
      A     M 221.2;
      A     M 203.4;
      AN    M 202.1;
      O     M 202.0;
      S     M 212.5;
      R     M 212.1;
      A     M 221.3;
      A     M 203.5;
      O     M 202.1;
      AN    M 202.0;
      S     M 212.1;
      R     M 212.5;
M004: NOP   0;
NETWORK
TITLE =
      AN    M 212.1;
      A     M 209.2;
      R     M 209.4;
      R     M 200.7;
      JC    M005;
      S     M 200.7;
      AN    M 212.1;
      S     M 209.2;
      A     M 212.1;
      R     M 209.2;
M005: A     M 209.4;
      =     M 202.5;
NETWORK
TITLE =
      AN    M 212.5;
      A     M 209.1;
      R     M 209.3;
      R     M 200.6;
      JC    M006;
      S     M 200.6;
      AN    M 212.5;
      S     M 209.1;
      A     M 212.5;
      R     M 209.1;
M006: A     M 209.3;
      =     M 202.4;
NETWORK
TITLE =
      A(;
      A     M 212.3;
      A     M 221.5;
      O;
      A     M 230.5;
      A     M 230.1;
      );
      A     M 203.5;
      A     M 209.0;
      =     M 200.5;
      =     #PARAM30;
      A(;
      A     M 212.2;
      A     M 221.5;
      O;
      A     M 230.4;
      A     M 230.1;
      );
      A     M 203.4;
      A     M 209.0;
      =     M 200.4;
      =     #PARAM21;
NETWORK
TITLE =
      A     M 230.0;
      A     M 230.1;
      O;
      A     M 221.5;
      A     #PARAM7;
      =     M 232.0;
      A     M 209.0;
      A     M 232.0;
      =     M 200.3;
      AN    M 209.0;
      A     M 232.0;
      =     M 200.2;
NETWORK
TITLE =
      A     M 200.7;
      A     M 202.2;
      =     M 203.7;
      A     M 200.6;
      A     M 202.3;
      =     M 203.6;
NETWORK
TITLE =
      A     M 202.5;
      O     M 202.4;
      O     M 203.7;
      O     M 203.6;
      =     M 200.0;
      A     M 202.5;
      O     M 203.7;
      =     M 201.5;
      A     M 202.4;
      O     M 203.6;
      =     M 201.2;
      A     M 200.7;
      AN    M 202.3;
      =     M 201.7;
      A     M 200.6;
      AN    M 202.2;
      =     M 201.4;
      A     M 200.7;
      A     M 202.3;
      =     M 201.6;
      A     M 200.6;
      A     M 202.2;
      =     M 201.3;
      A     M 209.0;
      =     M 201.1;
      AN    M 209.0;
      =     M 201.0;
NETWORK
TITLE =
      A     M 200.6;
      =     #PARAM24;
      A     M 200.7;
      =     #PARAM27;
      O(;
      A     "M 0.5";
      A     M 201.4;
      O;
      A     "M 1.6";
      A     M 201.2;
      O;
      O     M 201.3;
      O     M 221.4;
      );
      =     #PARAM31;
      A     M 201.0;
      O     M 221.4;
      =     #PARAM32;
      A     M 200.0;
      A     "M 1.6";
      O     M 200.1;
      O     M 221.4;
      =     #PARAM33;
      A     M 201.1;
      O     M 221.4;
      =     #PARAM34;
      O(;
      A     M 201.7;
      A     "M 0.5";
      O;
      A     M 201.5;
      A     "M 1.6";
      O;
      O     M 201.6;
      O     M 221.4;
      );
      =     #PARAM35;
      L     MW 200;
      T     DBW [AR1,P#6.0];
      L     MW 202;
      T     DBW [AR1,P#8.0];
      L     MW 208;
      T     DBW [AR1,P#12.0];
      L     MW 210;
      T     DBW [AR1,P#14.0];
      L     MB 212;
      T     DBW [AR1,P#16.0];
      L     MW 220;
      T     DBW [AR1,P#18.0];
      L     0;
      L     #PARAM20;
      ==I;
      JC    M009;
      T     MW 216;
      T     MW 240;
      L     MB 216;
      SLW   3;
      LAR1;
      L     DBW [AR1,P#0.0];
      T     MW 242;
      L     MW 240;
      SLW   12;
      SRW   12;
      T     MW 240;
      L     8;
      L     MB 241;
      >I;
      JC    M007;
      +     -8;
      SLW   8;
      INC   242;
      JU    M008;
M007: SLW   8;
      INC   243;
M008: T     MW 244;
      L     MB 244;
      L     MB 245;
      SLW   3;
      OW;
      LAR2;
      A     M 201.0;
      O     M 203.3;
      =     M [AR2,P#0.0];
      L     MB 217;
      SLW   3;
      LAR1;
      L     MW 242;
      T     DBW [AR1,P#0.0];
M009: L     0;
      L     #PARAM17;
      ==I;
      BEC;
      T     MW 222;
      L     MB 222;
      T     LW 10;
      OPN   DB [LW 10];
      L     MB 223;
      SLW   3;
      LAR1;
      L     MW 200;
      T     DBW [AR1,P#6.0];
      L     MW 202;
      T     DBW [AR1,P#8.0];
END_FUNCTION

FUNCTION "TE-VW2/2" : VOID	// FC 16
AUTHOR : SIMATIC
FAMILY : EA_DIS
NAME : TE_VW2_2
VERSION : 3.0
BEGIN
// (block stored without names or comments; labels and parameter names are numbered)
NETWORK
TITLE =
      L     0;
      L     #PARAM11;
      ==I;
      JC    M001;
      T     MW 212;
      L     MB 212;
      T     LW 10;
      OPN   DB [LW 10];
      L     MB 213;
      SLW   3;
      LAR1;
      L     DBW [AR1,P#0.0];
      T     MB 203;
M001: L     #PARAM9;
      T     MW 214;
      L     MB 214;
      T     LW 10;
      OPN   DB [LW 10];
      L     MB 215;
      SLW   3;
      LAR1;
      L     DBW [AR1,P#0.0];
      T     MW 200;
      L     DBW [AR1,P#2.0];
      T     MB 202;
      A     #PARAM1;
      =     M 200.0;
      A     #PARAM2;
      AN    M 201.7;
      =     M 204.5;
      A     #PARAM2;
      =     M 201.7;
      A     #PARAM3;
      AN    M 200.1;
      =     M 205.4;
      A     #PARAM3;
      =     M 200.1;
      A     #PARAM4;
      =     M 200.3;
      A     #PARAM5;
      AN    M 200.2;
      =     M 204.6;
      A     #PARAM5;
      =     M 200.2;
      A     #PARAM6;
      AN    M 200.4;
      =     M 205.5;
      A     #PARAM6;
      =     M 200.4;
      A     #PARAM7;
      =     M 201.6;
      A     #PARAM8;
      =     M 201.5;
NETWORK
TITLE =
      A     M 203.0;
      AN    M 202.0;
      =     M 204.0;
      A     M 203.0;
      =     M 202.0;
      A     M 203.1;
      AN    M 202.1;
      =     M 204.1;
      A     M 203.1;
      =     M 202.1;
NETWORK
TITLE =
      A(;
      A     M 205.4;
      A     M 201.6;
      O;
      A     M 204.0;
      AN    M 200.4;
      O;
      A     M 204.5;
      AN    M 200.4;
      AN    M 203.1;
      );
      A     M 200.0;
      =     M 202.5;
      A(;
      A     M 205.5;
      A     M 201.6;
      O;
      A     M 204.1;
      AN    M 200.1;
      O;
      A     M 204.6;
      AN    M 200.1;
      AN    M 203.0;
      );
      A     M 200.3;
      =     M 202.6;
NETWORK
TITLE =
      AN    M 201.1;
      S     M 201.0;
      A     "´1´";
      R     M 201.3;
      S     M 201.4;
NETWORK
TITLE =
      AN    M 201.0;
      JC    M002;
      A     M 202.6;
      S     M 201.1;
      R     M 201.0;
M002: NOP   0;
NETWORK
TITLE =
      AN    M 201.1;
      JC    M003;
      A     M 202.5;
      S     M 201.0;
      R     M 201.1;
M003: NOP   0;
NETWORK
TITLE =
      A     M 201.0;
      =     #PARAM12;
      A     M 201.1;
      =     #PARAM13;
      A     M 201.0;
      O     M 201.5;
      =     #PARAM14;
      A     M 201.1;
      O     M 201.5;
      =     #PARAM15;
      L     MW 200;
      T     DBW [AR1,P#0.0];
      L     MB 202;
      T     DBW [AR1,P#2.0];
      L     0;
      L     #PARAM10;
      ==I;
      BEC;
      T     MW 216;
      L     MB 216;
      T     LW 10;
      OPN   DB [LW 10];
      L     MB 217;
      SLW   3;
      LAR1;
      L     MB 201;
      T     DBW [AR1,P#0.0];
NETWORK
TITLE =
END_FUNCTION

FUNCTION "TE-VW2/1" : VOID	// FC 17
AUTHOR : SIMATIC
FAMILY : EA_DIS
NAME : TE_VW2_1
VERSION : 3.0
BEGIN
// (block stored without names or comments; labels and parameter names are numbered)
NETWORK
TITLE =
      L     0;
      L     #PARAM10;
      ==I;
      JC    M001;
      T     MW 212;
      L     MB 212;
      T     LW 10;
      OPN   DB [LW 10];
      L     MB 213;
      SLW   3;
      LAR1;
      L     DBW [AR1,P#0.0];
      T     MB 203;
M001: L     #PARAM8;
      T     MW 214;
      L     MB 214;
      T     LW 10;
      OPN   DB [LW 10];
      L     MB 215;
      SLW   3;
      LAR1;
      L     DBW [AR1,P#0.0];
      T     MW 200;
      L     DBW [AR1,P#2.0];
      T     MB 202;
      A     #PARAM1;
      =     M 200.0;
      A     #PARAM2;
      AN    M 201.7;
      =     M 204.5;
      A     #PARAM2;
      =     M 201.7;
      A     #PARAM3;
      AN    M 200.1;
      =     M 204.3;
      A     #PARAM3;
      =     M 200.1;
      A     #PARAM4;
      =     M 200.3;
      A     #PARAM5;
      AN    M 200.2;
      =     M 204.6;
      A     #PARAM5;
      =     M 200.2;
      A     #PARAM6;
      =     M 201.6;
      A     #PARAM7;
      =     M 201.5;
NETWORK
TITLE =
      A     M 203.0;
      AN    M 202.0;
      =     M 204.0;
      A     M 203.0;
      =     M 202.0;
NETWORK
TITLE =
      A     M 204.3;
      A     M 201.6;
      O;
      A     M 204.0;
      AN    M 200.1;
      =     M 202.5;
NETWORK
TITLE =
      AN    M 201.1;
      S     M 201.0;
      A     "´1´";
      R     M 201.3;
      R     M 201.4;
NETWORK
TITLE =
      AN    M 201.0;
      JC    M002;
      A     M 202.5;
      O     M 204.6;
      A     M 200.3;
      S     M 201.1;
      R     M 201.0;
      R     M 202.5;
M002: NOP   0;
NETWORK
TITLE =
      AN    M 201.1;
      JC    M003;
      A     M 202.5;
      O     M 204.5;
      A     M 200.0;
      S     M 201.0;
      R     M 201.1;
      R     M 202.5;
M003: NOP   0;
NETWORK
TITLE =
      A     M 201.0;
      =     #PARAM11;
      A     M 201.1;
      =     #PARAM12;
      A     M 201.0;
      O     M 201.5;
      =     #PARAM13;
      A     M 201.1;
      O     M 201.5;
      =     #PARAM14;
      L     MW 200;
      T     DBW [AR1,P#0.0];
      L     MB 202;
      T     DBW [AR1,P#2.0];
      L     0;
      L     #PARAM9;
      ==I;
      BEC;
      T     MW 216;
      L     MB 216;
      T     LW 10;
      OPN   DB [LW 10];
      L     MB 217;
      SLW   3;
      LAR1;
      L     MB 201;
      T     DBW [AR1,P#0.0];
NETWORK
TITLE =
END_FUNCTION

FUNCTION "TE_READ_RTM" : VOID	// FC 18
AUTHOR : SIMATIC
FAMILY : S7_300
NAME : TE_RTM
VERSION : 0.1
BEGIN
// (block stored without names or comments; labels and parameter names are numbered)
NETWORK
TITLE =
      OPN   #PARAM2;
      L     #PARAM3;
      T     MW 224;
      L     MB 225;
      SLW   3;
      LAR1;
      L     DBW [AR1,P#0.0];
      T     MW 210;
      L     DBW [AR1,P#2.0];
      T     MW 212;
      L     DBW [AR1,P#4.0];
      T     MW 214;
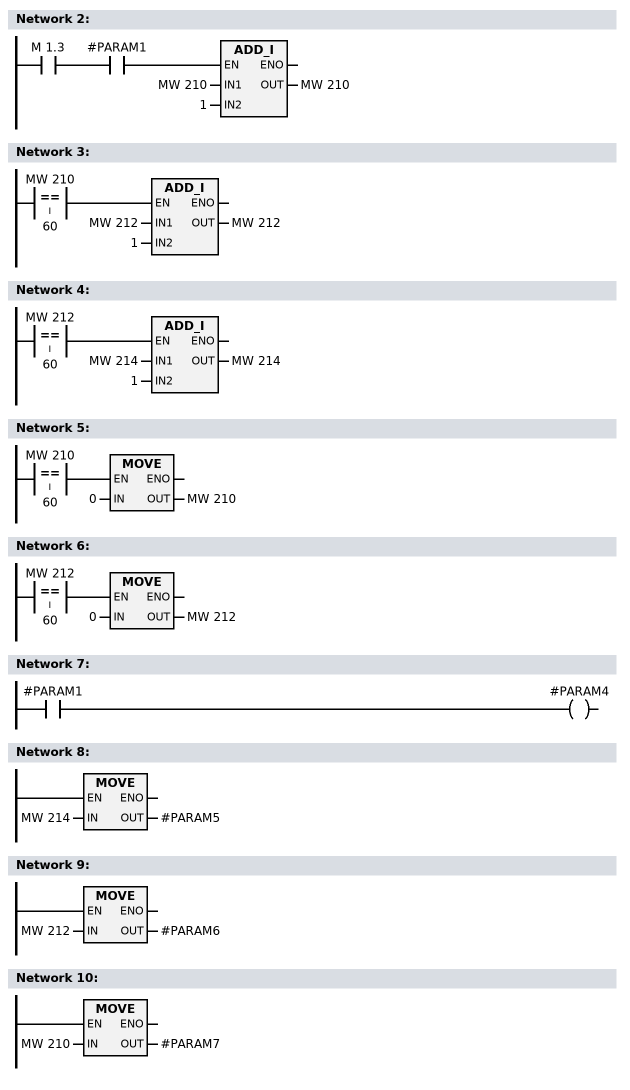
NETWORK
TITLE =
      A     "M 1.3";
      A     #PARAM1;
      JNB   M001;
      L     MW 210;
      L     1;
      +I;
      T     MW 210;
M001: NOP   0;
NETWORK
TITLE =
      A(;
      L     MW 210;
      L     60;
      ==I;
      );
      JNB   M002;
      L     MW 212;
      L     1;
      +I;
      T     MW 212;
M002: NOP   0;
NETWORK
TITLE =
      A(;
      L     MW 212;
      L     60;
      ==I;
      );
      JNB   M003;
      L     MW 214;
      L     1;
      +I;
      T     MW 214;
M003: NOP   0;
NETWORK
TITLE =
      A(;
      L     MW 210;
      L     60;
      ==I;
      );
      JNB   M004;
      L     0;
      T     MW 210;
M004: NOP   0;
NETWORK
TITLE =
      A(;
      L     MW 212;
      L     60;
      ==I;
      );
      JNB   M005;
      L     0;
      T     MW 212;
M005: NOP   0;
NETWORK
TITLE =
      A     #PARAM1;
      =     #PARAM4;
NETWORK
TITLE =
      L     MW 214;
      T     #PARAM5;
      NOP   0;
NETWORK
TITLE =
      L     MW 212;
      T     #PARAM6;
      NOP   0;
NETWORK
TITLE =
      L     MW 210;
      T     #PARAM7;
      NOP   0;
NETWORK
TITLE =
      L     MB 225;
      SLW   3;
      LAR1;
      T     DBW [AR1,P#0.0];
      L     MW 210;
      T     DBW [AR1,P#0.0];
      L     MW 212;
      T     DBW [AR1,P#2.0];
      L     MW 214;
      T     DBW [AR1,P#4.0];
END_FUNCTION

FUNCTION "TE-TAK" : VOID	// FC 29
AUTHOR : SIMATIC
FAMILY : EA_DIS
NAME : TE_TAKT
VERSION : 3.0
BEGIN
// (block stored without names or comments; labels and parameter names are numbered)
NETWORK
TITLE =
      OPN   #PARAM2;
      L     #PARAM1;
      L     0;
      <>I;
      JC    M005;
      L     DBB 33;
      T     MB 203;
      L     DBW 28;
      T     MW 200;
      A     M 201.0;
      S     M 203.0;
      L     MB 201;
      L     0;
      <>I;
      JC    M001;
      S     M 203.1;
      S     M 203.2;
      JU    M002;
M001: +     5;
      ==I;
      S     M 203.1;
      JU    M004;
M002: A     M 200.0;
      S     M 203.3;
      L     MB 200;
      L     0;
      <>I;
      JC    M003;
      S     M 203.6;
      S     M 203.5;
      JU    M004;
M003: +     30;
      <>I;
      JC    M004;
      S     M 203.5;
M004: L     MB 203;
      T     DBB 33;
      L     DBB 29;
      +     1;
      T     DBB 29;
      L     10;
      <I;
      BEC;
      L     0;
      T     DBB 29;
      L     DBB 28;
      +     1;
      T     DBB 28;
      L     60;
      <I;
      BEC;
      L     0;
      T     DBB 28;
      BEU;
M005: NOP   0;
NETWORK
TITLE =
// (network holds code this reader does not know; not shown)
NETWORK
TITLE =
      +     1;
      <>I;
      JC    M009;
      L     0;
      T     DBB 31;
M009: NOP   0;
NETWORK
TITLE =
END_FUNCTION

FUNCTION FC 30 : VOID
VERSION : 0.1
BEGIN
// (block stored without names or comments; labels and parameter names are numbered)
NETWORK
TITLE =
      L     0;
      <I;
      JC    M001;
      TAK;
      L     9;
      >I;
      JC    M001;
      TAK;
M001: L     4;
      *I;
      SLW   3;
      LAR1;
      OPN   DB 13;
      L     DBD [AR1,P#40.0];
      BEU;
NETWORK
TITLE =
      JL    M002;
      JU    M003;
      JU    M004;
      JU    M005;
      JU    M006;
      JU    M007;
      JU    M008;
      JU    M009;
      JU    M010;
      JU    M011;
      JU    M012;
M002: NOP   0;
M003: L     DB13.DBD 40;
      BEU;
M004: L     DB13.DBD 44;
      BEU;
M005: L     DB13.DBD 48;
      BEU;
M006: L     DB13.DBD 52;
      BEU;
M007: L     DB13.DBD 56;
      BEU;
M008: L     DB13.DBD 60;
      BEU;
M009: L     DB13.DBD 64;
      BEU;
M010: L     DB13.DBD 68;
      BEU;
M011: L     DB13.DBD 72;
      BEU;
M012: L     DB13.DBD 76;
      BEU;
END_FUNCTION

FUNCTION FC 31 : VOID
VERSION : 0.1
BEGIN
// (block stored without names or comments; labels and parameter names are numbered)
NETWORK
TITLE =
      JL    M001;
      JU    M002;
      JU    M003;
      JU    M004;
      JU    M005;
      JU    M006;
      JU    M007;
      JU    M008;
      JU    M009;
      JU    M010;
      JU    M011;
M001: NOP   0;
M002: L     DB13.DBD 0;
      BEU;
M003: L     DB13.DBD 4;
      BEU;
M004: L     DB13.DBD 8;
      BEU;
M005: L     DB13.DBD 12;
      BEU;
M006: L     DB13.DBD 16;
      BEU;
M007: L     DB13.DBD 20;
      BEU;
M008: L     DB13.DBD 24;
      BEU;
M009: L     DB13.DBD 28;
      BEU;
M010: L     DB13.DBD 32;
      BEU;
M011: L     DB13.DBD 36;
      BEU;
END_FUNCTION

FUNCTION FC 32 : VOID
VERSION : 0.1
BEGIN
// (block stored without names or comments; labels and parameter names are numbered)
NETWORK
TITLE =
      JL    M001;
      JU    M002;
      JU    M003;
      JU    M004;
      JU    M005;
      JU    M006;
      JU    M007;
      JU    M008;
      JU    M009;
      JU    M010;
      JU    M011;
M001: NOP   0;
M002: L     DB14.DBD 40;
      BEU;
M003: L     DB14.DBD 44;
      BEU;
M004: L     DB14.DBD 48;
      BEU;
M005: L     DB14.DBD 52;
      BEU;
M006: L     DB14.DBD 56;
      BEU;
M007: L     DB14.DBD 60;
      BEU;
M008: L     DB14.DBD 64;
      BEU;
M009: L     DB14.DBD 68;
      BEU;
M010: L     DB14.DBD 72;
      BEU;
M011: L     DB14.DBD 76;
      BEU;
END_FUNCTION

FUNCTION FC 33 : VOID
VERSION : 0.1
BEGIN
// (block stored without names or comments; labels and parameter names are numbered)
NETWORK
TITLE =
      JL    M001;
      JU    M002;
      JU    M003;
      JU    M004;
      JU    M005;
      JU    M006;
      JU    M007;
      JU    M008;
      JU    M009;
      JU    M010;
      JU    M011;
M001: NOP   0;
M002: L     DB14.DBD 0;
      BEU;
M003: L     DB14.DBD 4;
      BEU;
M004: L     DB14.DBD 8;
      BEU;
M005: L     DB14.DBD 12;
      BEU;
M006: L     DB14.DBD 16;
      BEU;
M007: L     DB14.DBD 20;
      BEU;
M008: L     DB14.DBD 24;
      BEU;
M009: L     DB14.DBD 28;
      BEU;
M010: L     DB14.DBD 32;
      BEU;
M011: L     DB14.DBD 36;
      BEU;
END_FUNCTION

FUNCTION "TE-GRENZ" : VOID	// FC 36
AUTHOR : SIMATIC
FAMILY : EA_DIS
NAME : TE_GRENZ
VERSION : 3.0
BEGIN
// (block stored without names or comments; labels and parameter names are numbered)
NETWORK
TITLE =
      AN    #PARAM4;
      R     #PARAM5;
      R     #PARAM6;
      BEC;
      L     #PARAM1;
      L     DW#16#0;
      ==R;
      JC    M001;
      L     #PARAM1;
      L     #PARAM2;
      >=R;
      S     #PARAM5;
      R     #PARAM6;
      BEC;
      L     #PARAM1;
      L     #PARAM3;
      <R;
M001: R     #PARAM5;
      S     #PARAM6;
NETWORK
TITLE =
END_FUNCTION

FUNCTION "TE-RETTEN" : VOID	// FC 38
AUTHOR : SIMATIC
FAMILY : EA_DIS
NAME : TE_RET
VERSION : 3.0
BEGIN
// (block stored without names or comments; labels and parameter names are numbered)
NETWORK
TITLE =
      OPN   #PARAM1;
      LAR1  P#DBX 0.0;
      LAR2  P#M 200.0;
      L     28;
M001: T     DBW 60;
      L     MW [AR2,P#0.0];
      T     DBW [AR1,P#0.0];
      +AR1  P#2.0;
      +AR2  P#2.0;
      L     DBW 60;
      LOOP  M001;
END_FUNCTION

FUNCTION "TE-LADEN" : VOID	// FC 39
AUTHOR : SIMATIC
FAMILY : EA_DIS
NAME : TE_LADEN
VERSION : 3.0
BEGIN
// (block stored without names or comments; labels and parameter names are numbered)
NETWORK
TITLE =
      OPN   #PARAM1;
      LAR1  P#DBX 0.0;
      LAR2  P#M 200.0;
      L     28;
M001: T     DBW 60;
      L     DBW [AR1,P#0.0];
      T     MW [AR2,P#0.0];
      +AR1  P#2.0;
      +AR2  P#2.0;
      L     DBW 60;
      LOOP  M001;
END_FUNCTION

FUNCTION FC 40 : VOID
VERSION : 0.1
BEGIN
// (block stored without names or comments; labels and parameter names are numbered)
NETWORK
TITLE =
      L     #PARAM4;
      L     #PARAM3;
      -R;
      T     LD 4;
      L     #PARAM2;
      L     #PARAM1;
      -R;
      T     LD 0;
      L     LD 4;
      /R;
      T     LD 8;
      L     #PARAM5;
      *R;
      T     LD 12;
      L     LD 8;
      L     #PARAM3;
      *R;
      T     LD 16;
      L     #PARAM1;
      L     LD 16;
      -R;
      L     LD 12;
      +R;
      T     #PARAM6;
END_FUNCTION

// FC 41: know-how protected block, not included

FUNCTION "TE-SCHALTER" : VOID	// FC 49
AUTHOR : SIMATIC
FAMILY : S7_300
NAME : ASL_MOD
VERSION : 0.0
BEGIN
// (block stored without names or comments; labels and parameter names are numbered)
NETWORK
TITLE =
      L     #PARAM2;
      T     MW 202;
      L     #PARAM3;
      T     MW 204;
      L     #PARAM4;
      T     MW 206;
      L     MB 202;
      T     LW 10;
      OPN   DB [LW 10];
      L     MB 203;
      SLW   3;
      LAR1;
      L     DBD [AR1,P#0.0];
      T     MD 210;
      AN    #PARAM1;
      JC    M001;
      L     MB 204;
      T     LW 10;
      OPN   DB [LW 10];
      L     MB 205;
      SLW   3;
      LAR1;
      L     DBD [AR1,P#0.0];
      T     MD 210;
M001: NOP   0;
      L     MB 206;
      T     LW 10;
      OPN   DB [LW 10];
      L     MB 207;
      SLW   3;
      LAR1;
      L     MD 210;
      T     DBD [AR1,P#0.0];
END_FUNCTION

FUNCTION FC 54 : VOID
AUTHOR : Elcard
FAMILY : Sinamics
NAME : Teleg370
VERSION : 0.0
BEGIN
// (block stored without names or comments; labels and parameter names are numbered)
NETWORK
TITLE =
      L     #PARAM1;
      T     LW 0;
      OPN   DB [LW 0];
      L     #PARAM2;
      ITD;
      SLD   3;
      T     LD 12;
      LAR1  P#L 2.0;
      L     B#16#10;
      T     LB [AR1,P#0.0];
      L     B#16#2;
      T     LB [AR1,P#1.0];
      L     10;
      T     LW [AR1,P#2.0];
      L     #PARAM1;
      T     LW [AR1,P#4.0];
      L     P#DBX 2.0;
      L     LD 12;
      +D;
      T     LD [AR1,P#6.0];
      L     P#DBX 0.0;
      L     LD 12;
      +D;
      LAR2;
NETWORK
TITLE =
      CALL  SFC 14 (
           $1                       := #PARAM3,
           $2                       := P#L 16.0,
           $3                       := P#L 2.0);
      L     LW 16;
      T     W [AR2,P#0.0];
NETWORK
TITLE =
      SET;
      =     DB201.DBX 14.2;
      A     #PARAM5;
      =     DB201.DBX 15.1;
      A     #PARAM5;
      A     DB201.DBX 3.4;
      AN    DB201.DBX 3.3;
      L     S5T#1S;
      SD    #PARAM6;
      A     #PARAM6;
      =     DB201.DBX 15.0;
      A     #PARAM4;
      =     DB201.DBX 15.7;
      A     DB201.DBX 3.6;
      =     #PARAM8;
      A     #PARAM4;
      R     #PARAM7;
      A     DB201.DBX 3.3;
      A     #PARAM5;
      S     #PARAM7;
NETWORK
TITLE =
      L     P#DBX 14.0;
      L     LD 12;
      +D;
      T     LD [AR1,P#6.0];
      CALL  SFC 15 (
           $1                       := #PARAM3,
           $2                       := P#L 2.0,
           $3                       := P#L 16.0);
      L     LW 16;
      T     W [AR2,P#12.0];
END_FUNCTION

FUNCTION FC 55 : VOID
AUTHOR : Elcard
FAMILY : Sinamics
NAME : Teleg370
VERSION : 0.0
BEGIN
// (block stored without names or comments; labels and parameter names are numbered)
NETWORK
TITLE =
      L     #PARAM1;
      T     LW 0;
      OPN   DB [LW 0];
      L     #PARAM2;
      ITD;
      SLD   3;
      T     LD 12;
      LAR1  P#L 2.0;
      L     B#16#10;
      T     LB [AR1,P#0.0];
      L     B#16#2;
      T     LB [AR1,P#1.0];
      L     4;
      T     LW [AR1,P#2.0];
      L     #PARAM1;
      T     LW [AR1,P#4.0];
      L     P#DBX 2.0;
      L     LD 12;
      +D;
      T     LD [AR1,P#6.0];
      L     P#DBX 0.0;
      L     LD 12;
      +D;
      LAR2;
NETWORK
TITLE =
      CALL  SFC 14 (
           $1                       := #PARAM3,
           $2                       := P#L 16.0,
           $3                       := P#L 2.0);
      L     LW 16;
      T     W [AR2,P#0.0];
NETWORK
TITLE =
      A     #PARAM4;
      A     DBX [AR2,P#3.3];
      =     DBX [AR2,P#9.7];
      A     DBX [AR2,P#3.3];
      =     #PARAM6;
      A     DBX [AR2,P#3.7];
      =     #PARAM5;
NETWORK
TITLE =
NETWORK
TITLE =
      L     P#DBX 6.0;
      L     LD 12;
      +D;
      T     LD [AR1,P#6.0];
      CALL  SFC 15 (
           $1                       := #PARAM3,
           $2                       := P#L 2.0,
           $3                       := P#L 16.0);
      L     LW 16;
      T     W [AR2,P#6.0];
END_FUNCTION

FUNCTION FC 56 : VOID
AUTHOR : Elcard
FAMILY : Sinamics
NAME : Teleg370
VERSION : 0.0
BEGIN
// (block stored without names or comments; labels and parameter names are numbered)
NETWORK
TITLE =
      L     #PARAM1;
      T     LW 0;
      OPN   DB [LW 0];
      L     #PARAM2;
      ITD;
      SLD   3;
      T     LD 12;
      LAR1  P#L 2.0;
      L     B#16#10;
      T     LB [AR1,P#0.0];
      L     B#16#2;
      T     LB [AR1,P#1.0];
      L     2;
      T     LW [AR1,P#2.0];
      L     #PARAM1;
      T     LW [AR1,P#4.0];
      L     P#DBX 2.0;
      L     LD 12;
      +D;
      T     LD [AR1,P#6.0];
      L     P#DBX 0.0;
      L     LD 12;
      +D;
      LAR2;
NETWORK
TITLE =
      CALL  SFC 14 (
           $1                       := #PARAM3,
           $2                       := P#L 16.0,
           $3                       := P#L 2.0);
      L     LW 16;
      T     W [AR2,P#0.0];
NETWORK
TITLE =
      SET;
      =     DB201.DBX 6.2;
      A     #PARAM5;
      =     DB201.DBX 7.1;
      A     #PARAM5;
      A     DB201.DBX 3.4;
      AN    DB201.DBX 3.3;
      L     S5T#1S;
      SD    #PARAM6;
      A     #PARAM6;
      =     DB201.DBX 7.0;
      A     #PARAM4;
      =     DB201.DBX 7.7;
      A     DB201.DBX 3.6;
      =     #PARAM8;
      A     #PARAM4;
      R     #PARAM7;
      A     DB201.DBX 3.3;
      A     #PARAM5;
      S     #PARAM7;
NETWORK
TITLE =
      L     P#DBX 6.0;
      L     LD 12;
      +D;
      T     LD [AR1,P#6.0];
      CALL  SFC 15 (
           $1                       := #PARAM3,
           $2                       := P#L 2.0,
           $3                       := P#L 16.0);
      L     LW 16;
      T     W [AR2,P#4.0];
END_FUNCTION

// FC 57: know-how protected block, not included

FUNCTION FC 58 : VOID
AUTHOR : Elcard
FAMILY : Inverter
NAME : Sinamics
VERSION : 0.1
BEGIN
// (block stored without names or comments; labels and parameter names are numbered)
NETWORK
TITLE =
      L     #PARAM1;
      T     LW 0;
      OPN   DB [LW 0];
      L     #PARAM2;
      ITD;
      SLD   3;
      T     LD 10;
      LAR1  P#L 0.0;
      L     B#16#10;
      T     LB [AR1,P#0.0];
      L     B#16#2;
      T     LB [AR1,P#1.0];
      L     #PARAM3;
      T     LW [AR1,P#2.0];
      L     #PARAM1;
      T     LW [AR1,P#4.0];
      L     P#DBX 2.0;
      L     LD 10;
      +D;
      T     LD [AR1,P#6.0];
      L     P#DBX 0.0;
      L     LD 10;
      +D;
      LAR2;
NETWORK
TITLE =
      CALL  SFC 14 (
           $1                       := #PARAM4,
           $2                       := P#L 14.0,
           $3                       := P#L 0.0);
      L     LW 14;
      T     W [AR2,P#0.0];
NETWORK
TITLE =
      A      [AR2,P#3.7];
      A     #PARAM5;
      =     #PARAM7;
      A      [AR2,P#3.3];
      A     DB201.DBX 3.2;
      A     #PARAM5;
      =     #PARAM6;
      AN    #PARAM6;
      AN    #PARAM7;
      =     #PARAM8;
END_FUNCTION

FUNCTION FC 59 : VOID
AUTHOR : Elcard
FAMILY : Inverter
NAME : Sinamics
VERSION : 0.2
BEGIN
// (block stored without names or comments; labels and parameter names are numbered)
NETWORK
TITLE =
      L     #PARAM1;
      T     LW 0;
      OPN   DB [LW 0];
      L     #PARAM2;
      ITD;
      SLD   3;
      T     LD 10;
      LAR1  P#L 0.0;
      L     B#16#10;
      T     LB [AR1,P#0.0];
      L     B#16#2;
      T     LB [AR1,P#1.0];
      L     #PARAM3;
      T     LW [AR1,P#2.0];
      L     #PARAM1;
      T     LW [AR1,P#4.0];
      L     P#DBX 2.0;
      L     LD 10;
      +D;
      T     LD [AR1,P#6.0];
      L     P#DBX 0.0;
      L     LD 10;
      +D;
      LAR2;
NETWORK
TITLE =
      O      [AR2,P#3.3];
      O      [AR2,P#3.7];
      A     #PARAM6;
      =      [AR2,P#23.7];
      A     #PARAM6;
      A      [AR2,P#14.7];
      =      [AR2,P#30.3];
      =      [AR2,P#30.7];
      A      [AR2,P#2.1];
      =      [AR2,P#22.2];
      A      [AR2,P#3.6];
      S      [AR2,P#23.5];
      S      [AR2,P#23.6];
      S      [AR2,P#28.0];
      A     #PARAM9;
      =      [AR2,P#23.1];
      AN    M 100.5;
      =      [AR2,P#23.4];
      AN    #PARAM7;
      =      [AR2,P#29.7];
      A      [AR2,P#3.3];
      R      [AR2,P#23.1];
      R      [AR2,P#23.2];
      R      [AR2,P#23.4];
      R      [AR2,P#23.5];
      R      [AR2,P#23.6];
      R      [AR2,P#28.0];
      R     #PARAM8;
      A     #PARAM5;
      =      [AR2,P#23.2];
      AN     [AR2,P#3.6];
      A      [AR2,P#3.5];
      A      [AR2,P#3.0];
      =      [AR2,P#23.3];
      A      [AR2,P#23.3];
      A     #PARAM8;
      =      [AR2,P#23.0];
NETWORK
TITLE =
      L     P#DBX 22.0;
      L     LD 10;
      +D;
      T     LD [AR1,P#6.0];
      CALL  SFC 15 (
           $1                       := #PARAM4,
           $2                       := P#L 0.0,
           $3                       := P#L 14.0);
      L     LW 14;
      T     W [AR2,P#42.0];
END_FUNCTION

FUNCTION FC 60 : VOID
AUTHOR : Elcard
FAMILY : Inverter
NAME : Sinamics
VERSION : 0.2
BEGIN
// (block stored without names or comments; labels and parameter names are numbered)
NETWORK
TITLE =
      L     #PARAM1;
      T     LW 0;
      OPN   DB [LW 0];
      L     #PARAM2;
      ITD;
      SLD   3;
      T     LD 10;
      LAR1  P#L 0.0;
      L     B#16#10;
      T     LB [AR1,P#0.0];
      L     B#16#2;
      T     LB [AR1,P#1.0];
      L     #PARAM3;
      T     LW [AR1,P#2.0];
      L     #PARAM1;
      T     LW [AR1,P#4.0];
      L     P#DBX 2.0;
      L     LD 10;
      +D;
      T     LD [AR1,P#6.0];
      L     P#DBX 0.0;
      L     LD 10;
      +D;
      LAR2;
NETWORK
TITLE =
      CALL  SFC 14 (
           $1                       := #PARAM4,
           $2                       := P#L 14.0,
           $3                       := P#L 0.0);
      L     LW 14;
      T     W [AR2,P#0.0];
NETWORK
TITLE =
      A      [AR2,P#3.7];
      A     #PARAM5;
      =     #PARAM7;
      A      [AR2,P#3.3];
      A     DB100.DBX 1.7;
      A     #PARAM5;
      S     #PARAM6;
      A     "M 7.7";
      R     #PARAM6;
      AN    #PARAM6;
      AN    #PARAM7;
      =     #PARAM8;
END_FUNCTION

FUNCTION FC 61 : VOID
AUTHOR : Elcard
FAMILY : Inverter
NAME : Sinamics
VERSION : 0.1
BEGIN
// (block stored without names or comments; labels and parameter names are numbered)
NETWORK
TITLE =
      L     #PARAM1;
      T     LW 0;
      OPN   DB [LW 0];
      L     #PARAM2;
      ITD;
      SLD   3;
      T     LD 10;
      LAR1  P#L 0.0;
      L     B#16#10;
      T     LB [AR1,P#0.0];
      L     B#16#2;
      T     LB [AR1,P#1.0];
      L     #PARAM3;
      T     LW [AR1,P#2.0];
      L     #PARAM1;
      T     LW [AR1,P#4.0];
      L     P#DBX 2.0;
      L     LD 10;
      +D;
      T     LD [AR1,P#6.0];
      L     P#DBX 0.0;
      L     LD 10;
      +D;
      LAR2;
NETWORK
TITLE =
      O      [AR2,P#3.3];
      O      [AR2,P#3.7];
      A     #PARAM6;
      =      [AR2,P#23.7];
      A      [AR2,P#2.1];
      =      [AR2,P#22.2];
      A      [AR2,P#3.6];
      S      [AR2,P#23.5];
      S      [AR2,P#23.6];
      S      [AR2,P#23.4];
      A     #PARAM9;
      =      [AR2,P#23.1];
      AN    #PARAM7;
      =      [AR2,P#29.7];
      A      [AR2,P#3.3];
      R      [AR2,P#23.1];
      R      [AR2,P#23.2];
      R      [AR2,P#23.4];
      R      [AR2,P#23.5];
      R      [AR2,P#23.6];
      R     #PARAM8;
      A     #PARAM5;
      =      [AR2,P#23.2];
      AN     [AR2,P#3.6];
      A      [AR2,P#3.5];
      A      [AR2,P#3.0];
      =      [AR2,P#23.3];
      A      [AR2,P#23.3];
      A     #PARAM8;
      =      [AR2,P#23.0];
NETWORK
TITLE =
      L     P#DBX 22.0;
      L     LD 10;
      +D;
      T     LD [AR1,P#6.0];
      CALL  SFC 15 (
           $1                       := #PARAM4,
           $2                       := P#L 0.0,
           $3                       := P#L 14.0);
      L     LW 14;
      T     W [AR2,P#42.0];
END_FUNCTION

